// TIA Portal V17 export
// export: Created 2023-04-04T13:27:31.7395928Z, ExportSetting WithDefaults, DisplayName Totally Integrated Automation Portal, DisplayVersion V17, DisplayName TIA Portal Openness, DisplayVersion V17, DisplayName TIA Portal Version Control Interface, DisplayVersion V17, DisplayName STEP 7 Professional, DisplayVersion V17, DisplayName STEP 7 Safety, DisplayVersion V17, DisplayName WinCC Advanced, DisplayVersion V17
TYPE "typ_Workpiece"
// stored: IsFailsafeCompliant false
   STRUCT
      s_id : String;
      s_type : String;
      s_state : String;
   END_STRUCT;
END_TYPE
